{attribute 'GeneratedUsingTerminal: EJ7334-0008-0016'}
{attribute addProperty BoxType "EJ7334-0008-0016"}
{attribute addProperty Id "EnableBOOL1ResetBOOL1"}
{attribute addProperty CRC "4284135858"}
{attribute addProperty Size "2"}
TYPE Control_FF5AB9B2 :
STRUCT
	{attribute addProperty Name "Enable"}
	Enable : BOOL;
	{attribute addProperty Name "Reset"}
	Reset : BOOL;
END_STRUCT
END_TYPE

(* stored: Version 1.2.0.0, ProductVersion 3.1.4024.9
   DUT Control_FF5AB9B2: Id {f594c19d-fe11-4726-906e-6065795100dc} *)
